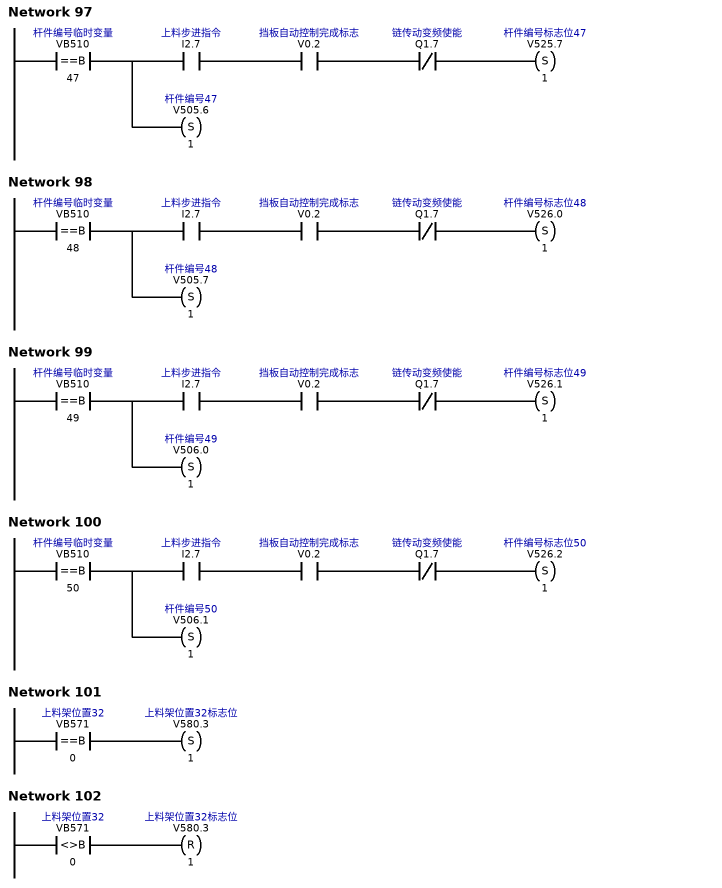
[picture p48: SBR17 networks 97-102]
Network 97
LDB=   杆件编号临时变量:VB510, 47
LPS
A      上料步进指令:I2.7
A      挡板自动控制完成标志:V0.2
AN     链传动变频使能:Q1.7
S      杆件编号标志位47:V525.7, 1
LPP
S      杆件编号47:V505.6, 1
Network 98
LDB=   杆件编号临时变量:VB510, 48
LPS
A      上料步进指令:I2.7
A      挡板自动控制完成标志:V0.2
AN     链传动变频使能:Q1.7
S      杆件编号标志位48:V526.0, 1
LPP
S      杆件编号48:V505.7, 1
Network 99
LDB=   杆件编号临时变量:VB510, 49
LPS
A      上料步进指令:I2.7
A      挡板自动控制完成标志:V0.2
AN     链传动变频使能:Q1.7
S      杆件编号标志位49:V526.1, 1
LPP
S      杆件编号49:V506.0, 1
Network 100
LDB=   杆件编号临时变量:VB510, 50
LPS
A      上料步进指令:I2.7
A      挡板自动控制完成标志:V0.2
AN     链传动变频使能:Q1.7
S      杆件编号标志位50:V526.2, 1
LPP
S      杆件编号50:V506.1, 1
Network 101
LDB=   上料架位置32:VB571, 0
S      上料架位置32标志位:V580.3, 1
Network 102
LDB<>  上料架位置32:VB571, 0
R      上料架位置32标志位:V580.3, 1
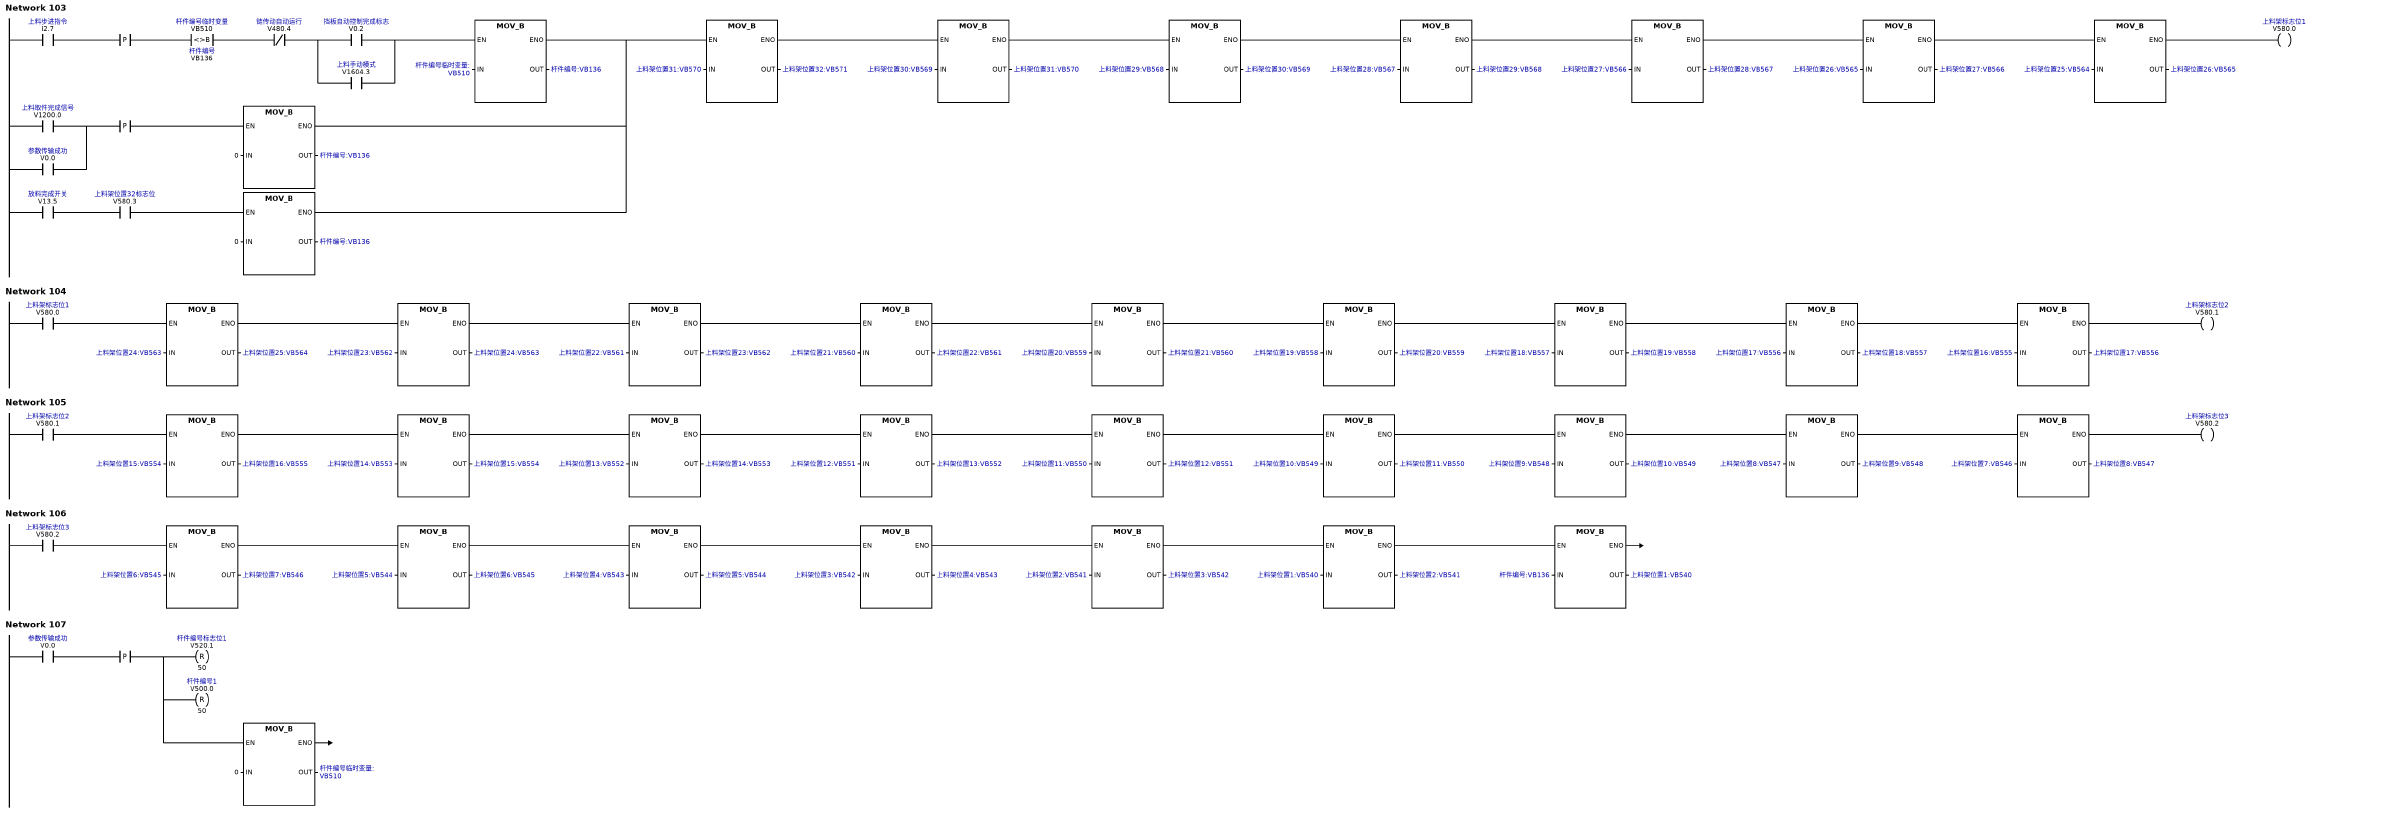
Network 103
LD     上料步进指令:I2.7
EU
AB<>   杆件编号临时变量:VB510, 杆件编号:VB136
AN     链传动自动运行:V480.4
LD     挡板自动控制完成标志:V0.2
O      上料手动模式:V1604.3
ALD
MOVB   杆件编号临时变量:VB510, 杆件编号:VB136
AENO
LD     上料取件完成信号:V1200.0
O      参数传输成功:V0.0
EU
MOVB   0, 杆件编号:VB136
AENO
OLD
LD     放料完成开关:V13.5
A      上料架位置32标志位:V580.3
MOVB   0, 杆件编号:VB136
AENO
OLD
MOVB   上料架位置31:VB570, 上料架位置32:VB571
AENO
MOVB   上料架位置30:VB569, 上料架位置31:VB570
AENO
MOVB   上料架位置29:VB568, 上料架位置30:VB569
AENO
MOVB   上料架位置28:VB567, 上料架位置29:VB568
AENO
MOVB   上料架位置27:VB566, 上料架位置28:VB567
AENO
MOVB   上料架位置26:VB565, 上料架位置27:VB566
AENO
MOVB   上料架位置25:VB564, 上料架位置26:VB565
AENO
=      上料架标志位1:V580.0
Network 104
LD     上料架标志位1:V580.0
MOVB   上料架位置24:VB563, 上料架位置25:VB564
AENO
MOVB   上料架位置23:VB562, 上料架位置24:VB563
AENO
MOVB   上料架位置22:VB561, 上料架位置23:VB562
AENO
MOVB   上料架位置21:VB560, 上料架位置22:VB561
AENO
MOVB   上料架位置20:VB559, 上料架位置21:VB560
AENO
MOVB   上料架位置19:VB558, 上料架位置20:VB559
AENO
MOVB   上料架位置18:VB557, 上料架位置19:VB558
AENO
MOVB   上料架位置17:VB556, 上料架位置18:VB557
AENO
MOVB   上料架位置16:VB555, 上料架位置17:VB556
AENO
=      上料架标志位2:V580.1
Network 105
LD     上料架标志位2:V580.1
MOVB   上料架位置15:VB554, 上料架位置16:VB555
AENO
MOVB   上料架位置14:VB553, 上料架位置15:VB554
AENO
MOVB   上料架位置13:VB552, 上料架位置14:VB553
AENO
MOVB   上料架位置12:VB551, 上料架位置13:VB552
AENO
MOVB   上料架位置11:VB550, 上料架位置12:VB551
AENO
MOVB   上料架位置10:VB549, 上料架位置11:VB550
AENO
MOVB   上料架位置9:VB548, 上料架位置10:VB549
AENO
MOVB   上料架位置8:VB547, 上料架位置9:VB548
AENO
MOVB   上料架位置7:VB546, 上料架位置8:VB547
AENO
=      上料架标志位3:V580.2
Network 106
LD     上料架标志位3:V580.2
MOVB   上料架位置6:VB545, 上料架位置7:VB546
AENO
MOVB   上料架位置5:VB544, 上料架位置6:VB545
AENO
MOVB   上料架位置4:VB543, 上料架位置5:VB544
AENO
MOVB   上料架位置3:VB542, 上料架位置4:VB543
AENO
MOVB   上料架位置2:VB541, 上料架位置3:VB542
AENO
MOVB   上料架位置1:VB540, 上料架位置2:VB541
AENO
MOVB   杆件编号:VB136, 上料架位置1:VB540
Network 107
LD     参数传输成功:V0.0
EU
R      杆件编号标志位1:V520.1, 50
R      杆件编号1:V500.0, 50
MOVB   0, 杆件编号临时变量:VB510
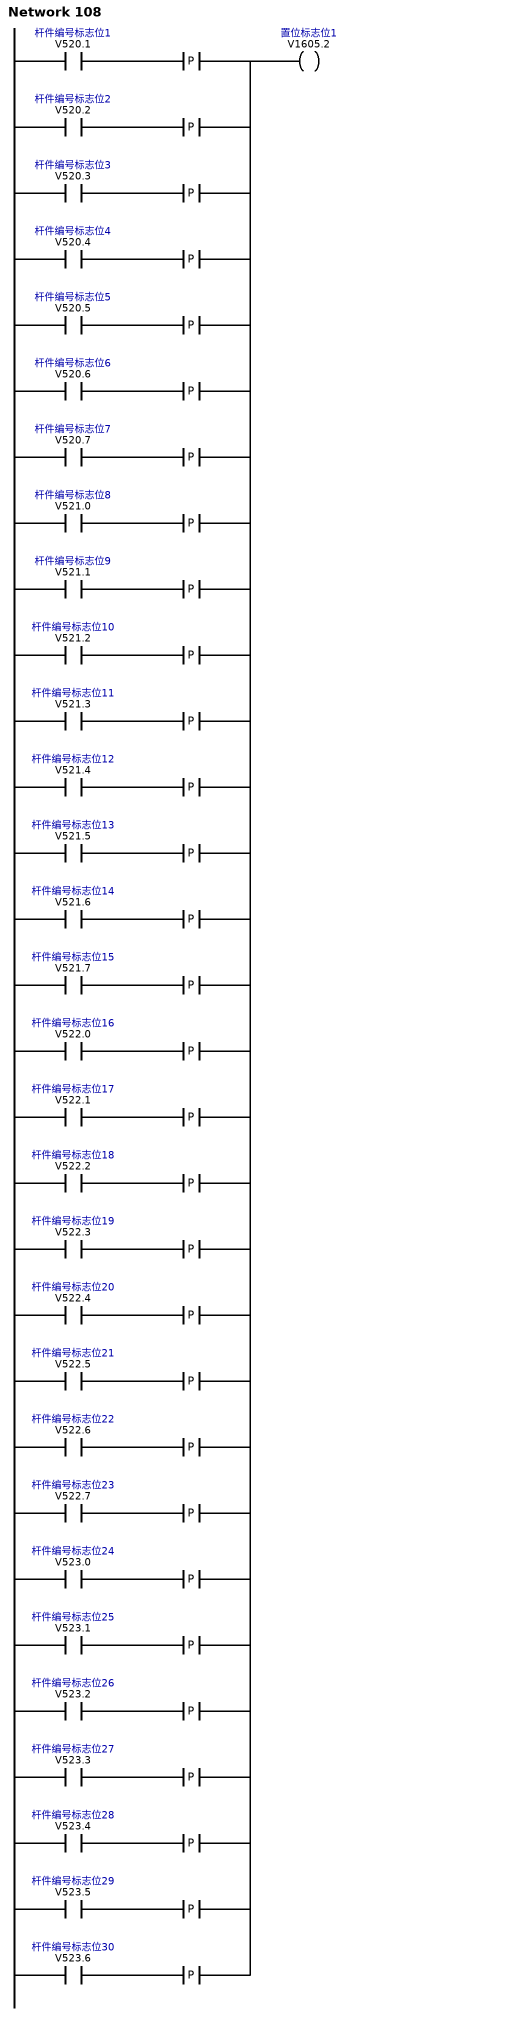
Network 108
LD     杆件编号标志位1:V520.1
EU
LD     杆件编号标志位2:V520.2
EU
OLD
LD     杆件编号标志位3:V520.3
EU
OLD
LD     杆件编号标志位4:V520.4
EU
OLD
LD     杆件编号标志位5:V520.5
EU
OLD
LD     杆件编号标志位6:V520.6
EU
OLD
LD     杆件编号标志位7:V520.7
EU
OLD
LD     杆件编号标志位8:V521.0
EU
OLD
LD     杆件编号标志位9:V521.1
EU
OLD
LD     杆件编号标志位10:V521.2
EU
OLD
LD     杆件编号标志位11:V521.3
EU
OLD
LD     杆件编号标志位12:V521.4
EU
OLD
LD     杆件编号标志位13:V521.5
EU
OLD
LD     杆件编号标志位14:V521.6
EU
OLD
LD     杆件编号标志位15:V521.7
EU
OLD
LD     杆件编号标志位16:V522.0
EU
OLD
LD     杆件编号标志位17:V522.1
EU
OLD
LD     杆件编号标志位18:V522.2
EU
OLD
LD     杆件编号标志位19:V522.3
EU
OLD
LD     杆件编号标志位20:V522.4
EU
OLD
LD     杆件编号标志位21:V522.5
EU
OLD
LD     杆件编号标志位22:V522.6
EU
OLD
LD     杆件编号标志位23:V522.7
EU
OLD
LD     杆件编号标志位24:V523.0
EU
OLD
LD     杆件编号标志位25:V523.1
EU
OLD
LD     杆件编号标志位26:V523.2
EU
OLD
LD     杆件编号标志位27:V523.3
EU
OLD
LD     杆件编号标志位28:V523.4
EU
OLD
LD     杆件编号标志位29:V523.5
EU
OLD
LD     杆件编号标志位30:V523.6
EU
OLD
=      置位标志位1:V1605.2
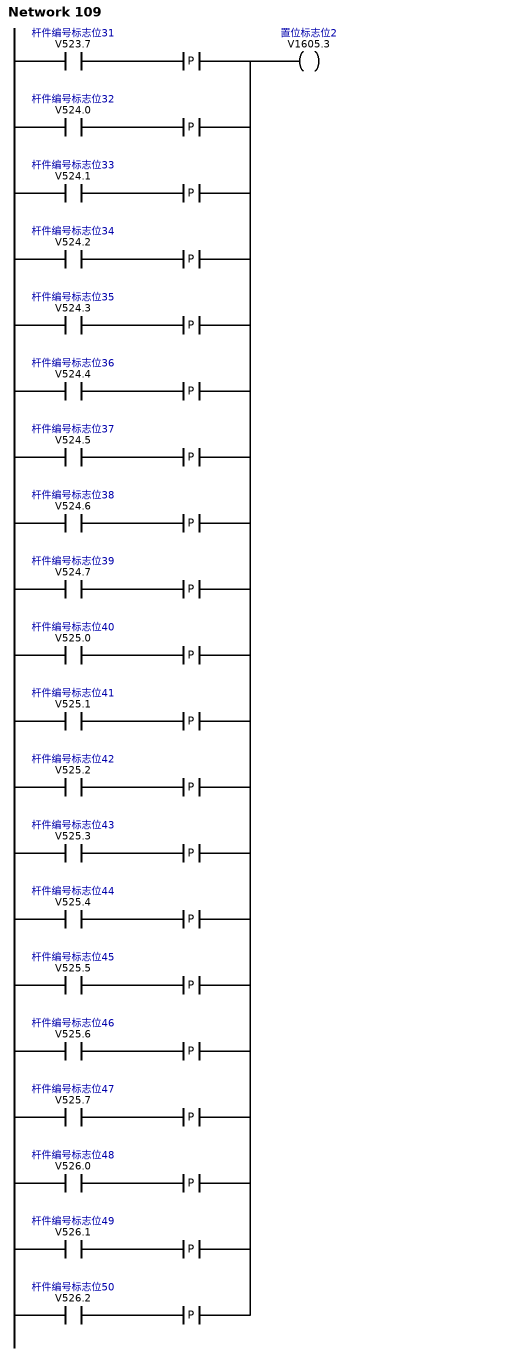
Network 109
LD     杆件编号标志位31:V523.7
EU
LD     杆件编号标志位32:V524.0
EU
OLD
LD     杆件编号标志位33:V524.1
EU
OLD
LD     杆件编号标志位34:V524.2
EU
OLD
LD     杆件编号标志位35:V524.3
EU
OLD
LD     杆件编号标志位36:V524.4
EU
OLD
LD     杆件编号标志位37:V524.5
EU
OLD
LD     杆件编号标志位38:V524.6
EU
OLD
LD     杆件编号标志位39:V524.7
EU
OLD
LD     杆件编号标志位40:V525.0
EU
OLD
LD     杆件编号标志位41:V525.1
EU
OLD
LD     杆件编号标志位42:V525.2
EU
OLD
LD     杆件编号标志位43:V525.3
EU
OLD
LD     杆件编号标志位44:V525.4
EU
OLD
LD     杆件编号标志位45:V525.5
EU
OLD
LD     杆件编号标志位46:V525.6
EU
OLD
LD     杆件编号标志位47:V525.7
EU
OLD
LD     杆件编号标志位48:V526.0
EU
OLD
LD     杆件编号标志位49:V526.1
EU
OLD
LD     杆件编号标志位50:V526.2
EU
OLD
=      置位标志位2:V1605.3
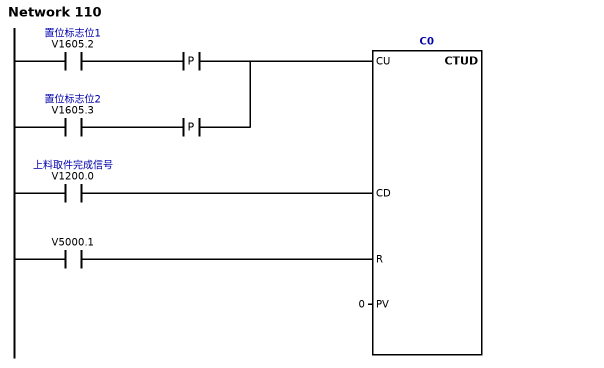
Network 110
LD     置位标志位1:V1605.2
EU
LD     置位标志位2:V1605.3
EU
OLD
LD     上料取件完成信号:V1200.0
LD     V5000.1
CTUD   C0, 0
END_SUBROUTINE_BLOCK

SUBROUTINE_BLOCK 冷却电机手动控制:SBR18
TITLE=子程序注释
BEGIN
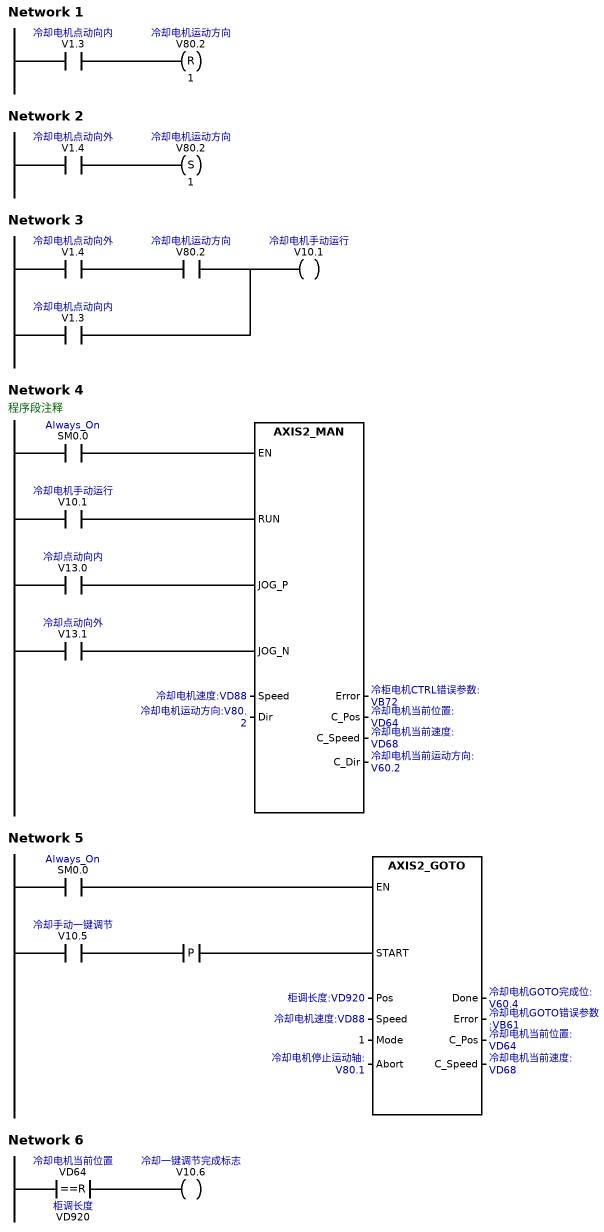
Network 1
LD     冷却电机点动向内:V1.3
R      冷却电机运动方向:V80.2, 1
Network 2
LD     冷却电机点动向外:V1.4
S      冷却电机运动方向:V80.2, 1
Network 3
LD     冷却电机点动向外:V1.4
A      冷却电机运动方向:V80.2
O      冷却电机点动向内:V1.3
=      冷却电机手动运行:V10.1
Network 4
// 程序段注释
LD     Always_On:SM0.0
=      L60.0
LD     冷却电机手动运行:V10.1
=      L63.7
LD     冷却点动向内:V13.0
=      L63.6
LD     冷却点动向外:V13.1
=      L63.5
LD     L60.0
CALL   AXIS2_MAN:SBR11, L63.7, L63.6, L63.5, 冷却电机速度:VD88, 冷却电机运动方向:V80.2, 冷柜电机CTRL错误参数:VB72, 冷却电机当前位置:VD64, 冷却电机当前速度:VD68, 冷却电机当前运动方向:V60.2
Network 5
LD     Always_On:SM0.0
=      L60.0
LD     冷却手动一键调节:V10.5
EU
=      L63.7
LD     L60.0
CALL   AXIS2_GOTO:SBR12, L63.7, 柜调长度:VD920, 冷却电机速度:VD88, 1, 冷却电机停止运动轴:V80.1, 冷却电机GOTO完成位:V60.4, 冷却电机GOTO错误参数:VB61, 冷却电机当前位置:VD64, 冷却电机当前速度:VD68
Network 6
LDR=   冷却电机当前位置:VD64, 柜调长度:VD920
=      冷却一键调节完成标志:V10.6
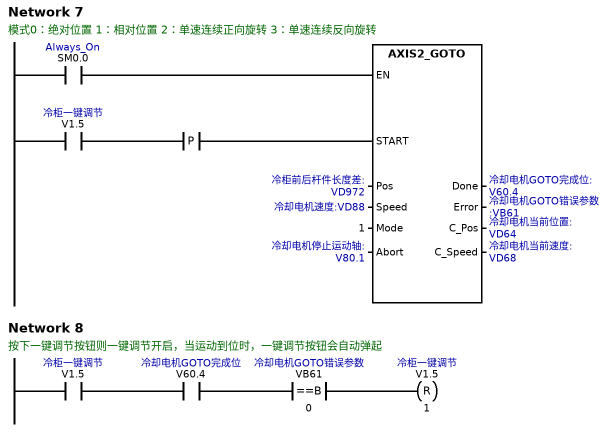
Network 7
// 模式0：绝对位置 1：相对位置 2：单速连续正向旋转 3：单速连续反向旋转
LD     Always_On:SM0.0
=      L60.0
LD     冷柜一键调节:V1.5
EU
=      L63.7
LD     L60.0
CALL   AXIS2_GOTO:SBR12, L63.7, 冷柜前后杆件长度差:VD972, 冷却电机速度:VD88, 1, 冷却电机停止运动轴:V80.1, 冷却电机GOTO完成位:V60.4, 冷却电机GOTO错误参数:VB61, 冷却电机当前位置:VD64, 冷却电机当前速度:VD68
Network 8
// 按下一键调节按钮则一键调节开启，当运动到位时，一键调节按钮会自动弹起
LD     冷柜一键调节:V1.5
A      冷却电机GOTO完成位:V60.4
AB=    冷却电机GOTO错误参数:VB61, 0
R      冷柜一键调节:V1.5, 1
END_SUBROUTINE_BLOCK

SUBROUTINE_BLOCK 链传动电机控制:SBR19
TITLE=子程序注释
BEGIN
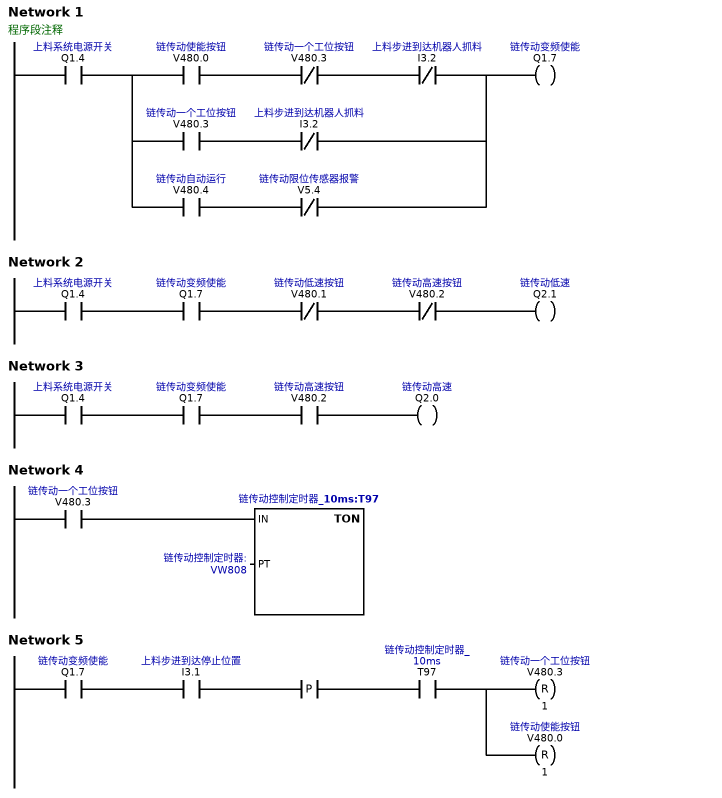
Network 1
// 程序段注释
LD     上料系统电源开关:Q1.4
LD     链传动使能按钮:V480.0
AN     链传动一个工位按钮:V480.3
AN     上料步进到达机器人抓料:I3.2
LD     链传动一个工位按钮:V480.3
AN     上料步进到达机器人抓料:I3.2
OLD
LD     链传动自动运行:V480.4
AN     链传动限位传感器报警:V5.4
OLD
ALD
=      链传动变频使能:Q1.7
Network 2
LD     上料系统电源开关:Q1.4
A      链传动变频使能:Q1.7
AN     链传动低速按钮:V480.1
AN     链传动高速按钮:V480.2
=      链传动低速:Q2.1
Network 3
LD     上料系统电源开关:Q1.4
A      链传动变频使能:Q1.7
A      链传动高速按钮:V480.2
=      链传动高速:Q2.0
Network 4
LD     链传动一个工位按钮:V480.3
TON    链传动控制定时器_10ms:T97, 链传动控制定时器:VW808
Network 5
LD     链传动变频使能:Q1.7
A      上料步进到达停止位置:I3.1
EU
A      链传动控制定时器_10ms:T97
R      链传动一个工位按钮:V480.3, 1
R      链传动使能按钮:V480.0, 1
END_SUBROUTINE_BLOCK

SUBROUTINE_BLOCK 数据初始化:SBR20
TITLE=子程序注释
BEGIN
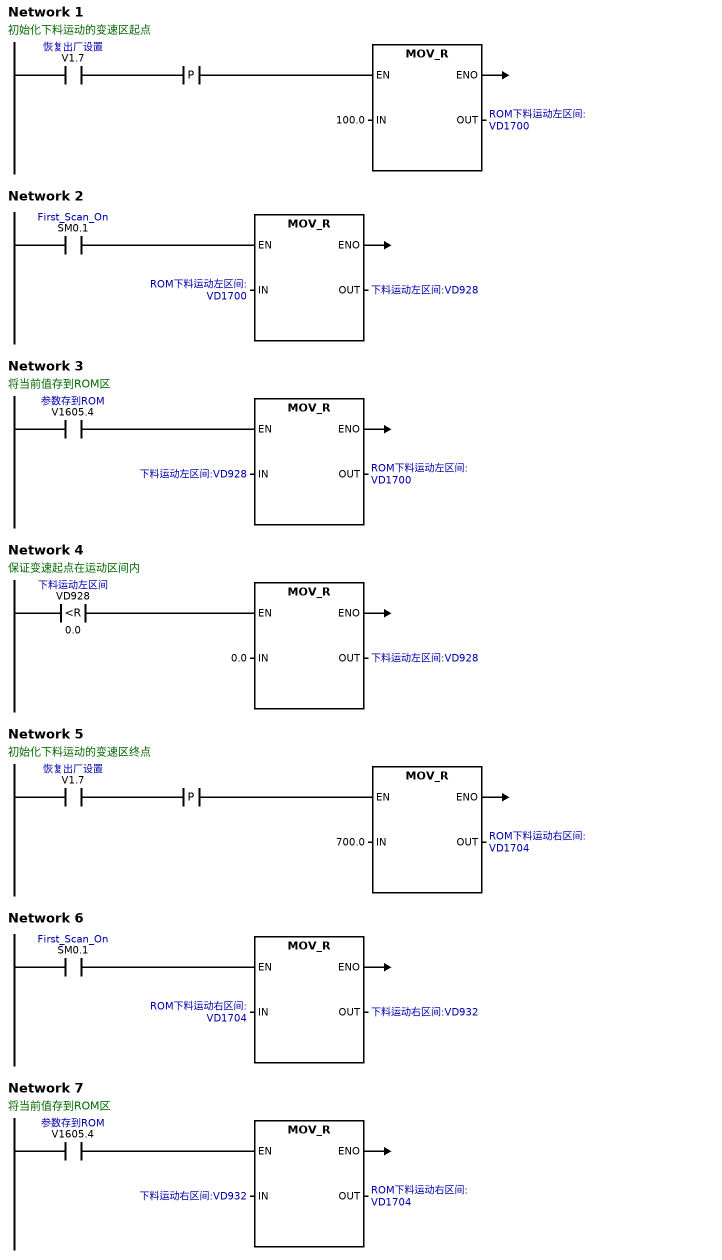
Network 1
// 初始化下料运动的变速区起点
LD     恢复出厂设置:V1.7
EU
MOVR   100.0, ROM下料运动左区间:VD1700
Network 2
LD     First_Scan_On:SM0.1
MOVR   ROM下料运动左区间:VD1700, 下料运动左区间:VD928
Network 3
// 将当前值存到ROM区
LD     参数存到ROM:V1605.4
MOVR   下料运动左区间:VD928, ROM下料运动左区间:VD1700
Network 4
// 保证变速起点在运动区间内
LDR<   下料运动左区间:VD928, 0.0
MOVR   0.0, 下料运动左区间:VD928
Network 5
// 初始化下料运动的变速区终点
LD     恢复出厂设置:V1.7
EU
MOVR   700.0, ROM下料运动右区间:VD1704
Network 6
LD     First_Scan_On:SM0.1
MOVR   ROM下料运动右区间:VD1704, 下料运动右区间:VD932
Network 7
// 将当前值存到ROM区
LD     参数存到ROM:V1605.4
MOVR   下料运动右区间:VD932, ROM下料运动右区间:VD1704
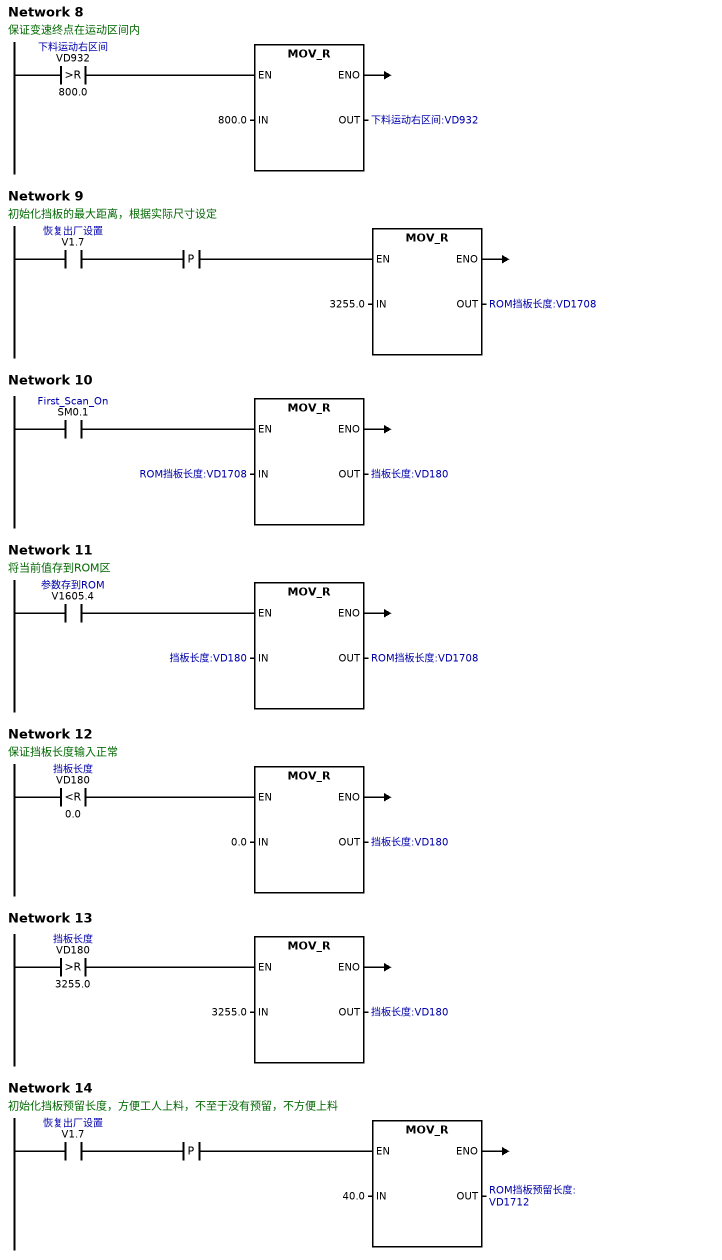
Network 8
// 保证变速终点在运动区间内
LDR>   下料运动右区间:VD932, 800.0
MOVR   800.0, 下料运动右区间:VD932
Network 9
// 初始化挡板的最大距离，根据实际尺寸设定
LD     恢复出厂设置:V1.7
EU
MOVR   3255.0, ROM挡板长度:VD1708
Network 10
LD     First_Scan_On:SM0.1
MOVR   ROM挡板长度:VD1708, 挡板长度:VD180
Network 11
// 将当前值存到ROM区
LD     参数存到ROM:V1605.4
MOVR   挡板长度:VD180, ROM挡板长度:VD1708
Network 12
// 保证挡板长度输入正常
LDR<   挡板长度:VD180, 0.0
MOVR   0.0, 挡板长度:VD180
Network 13
LDR>   挡板长度:VD180, 3255.0
MOVR   3255.0, 挡板长度:VD180
Network 14
// 初始化挡板预留长度，方便工人上料，不至于没有预留，不方便上料
LD     恢复出厂设置:V1.7
EU
MOVR   40.0, ROM挡板预留长度:VD1712
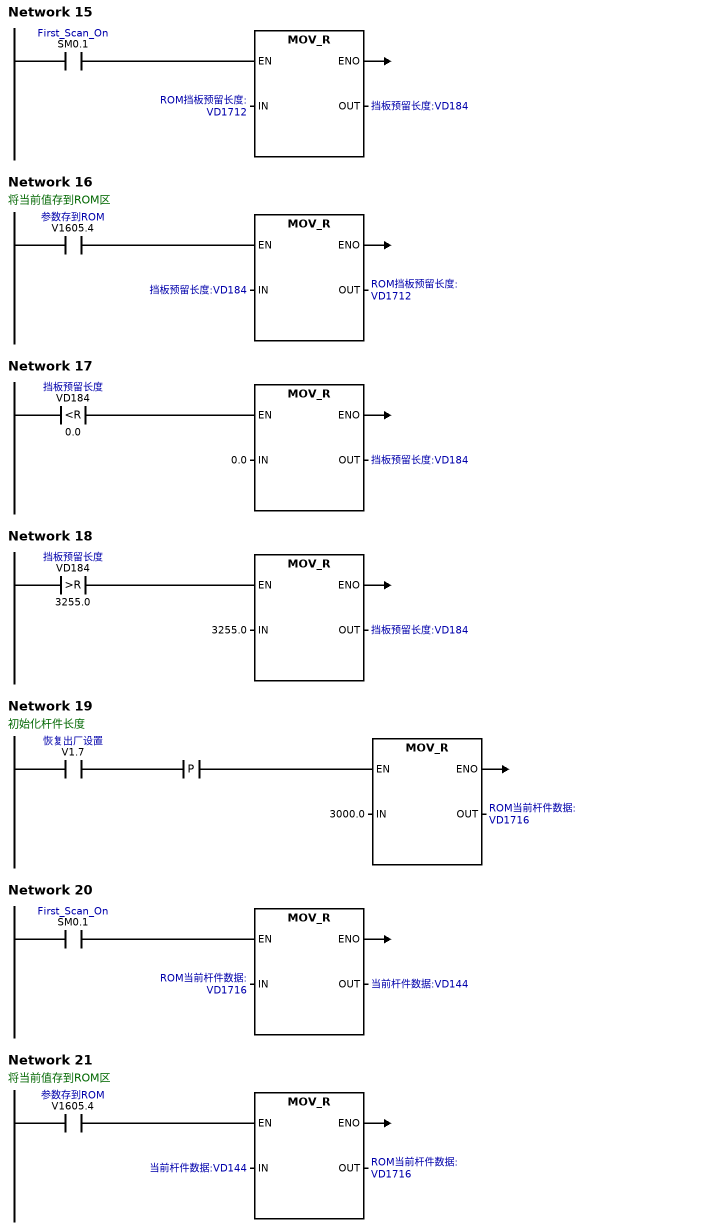
Network 15
LD     First_Scan_On:SM0.1
MOVR   ROM挡板预留长度:VD1712, 挡板预留长度:VD184
Network 16
// 将当前值存到ROM区
LD     参数存到ROM:V1605.4
MOVR   挡板预留长度:VD184, ROM挡板预留长度:VD1712
Network 17
LDR<   挡板预留长度:VD184, 0.0
MOVR   0.0, 挡板预留长度:VD184
Network 18
LDR>   挡板预留长度:VD184, 3255.0
MOVR   3255.0, 挡板预留长度:VD184
Network 19
// 初始化杆件长度
LD     恢复出厂设置:V1.7
EU
MOVR   3000.0, ROM当前杆件数据:VD1716
Network 20
LD     First_Scan_On:SM0.1
MOVR   ROM当前杆件数据:VD1716, 当前杆件数据:VD144
Network 21
// 将当前值存到ROM区
LD     参数存到ROM:V1605.4
MOVR   当前杆件数据:VD144, ROM当前杆件数据:VD1716
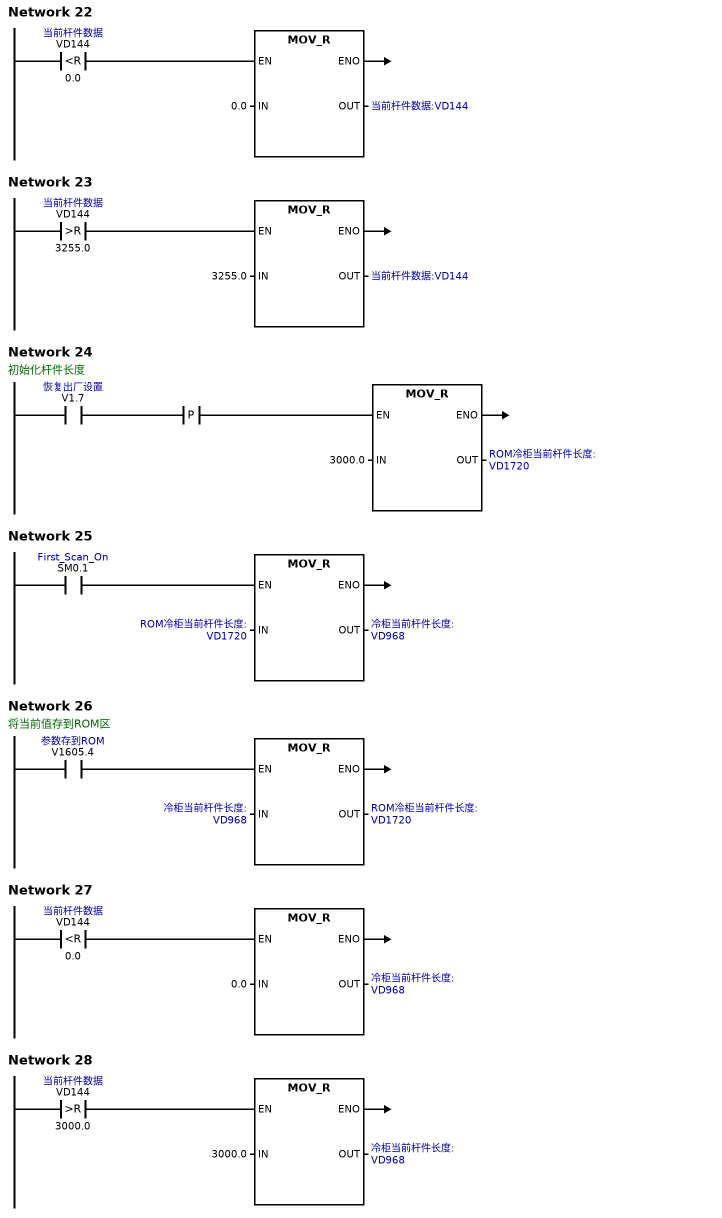
Network 22
LDR<   当前杆件数据:VD144, 0.0
MOVR   0.0, 当前杆件数据:VD144
Network 23
LDR>   当前杆件数据:VD144, 3255.0
MOVR   3255.0, 当前杆件数据:VD144
Network 24
// 初始化杆件长度
LD     恢复出厂设置:V1.7
EU
MOVR   3000.0, ROM冷柜当前杆件长度:VD1720
Network 25
LD     First_Scan_On:SM0.1
MOVR   ROM冷柜当前杆件长度:VD1720, 冷柜当前杆件长度:VD968
Network 26
// 将当前值存到ROM区
LD     参数存到ROM:V1605.4
MOVR   冷柜当前杆件长度:VD968, ROM冷柜当前杆件长度:VD1720
Network 27
LDR<   当前杆件数据:VD144, 0.0
MOVR   0.0, 冷柜当前杆件长度:VD968
Network 28
LDR>   当前杆件数据:VD144, 3000.0
MOVR   3000.0, 冷柜当前杆件长度:VD968
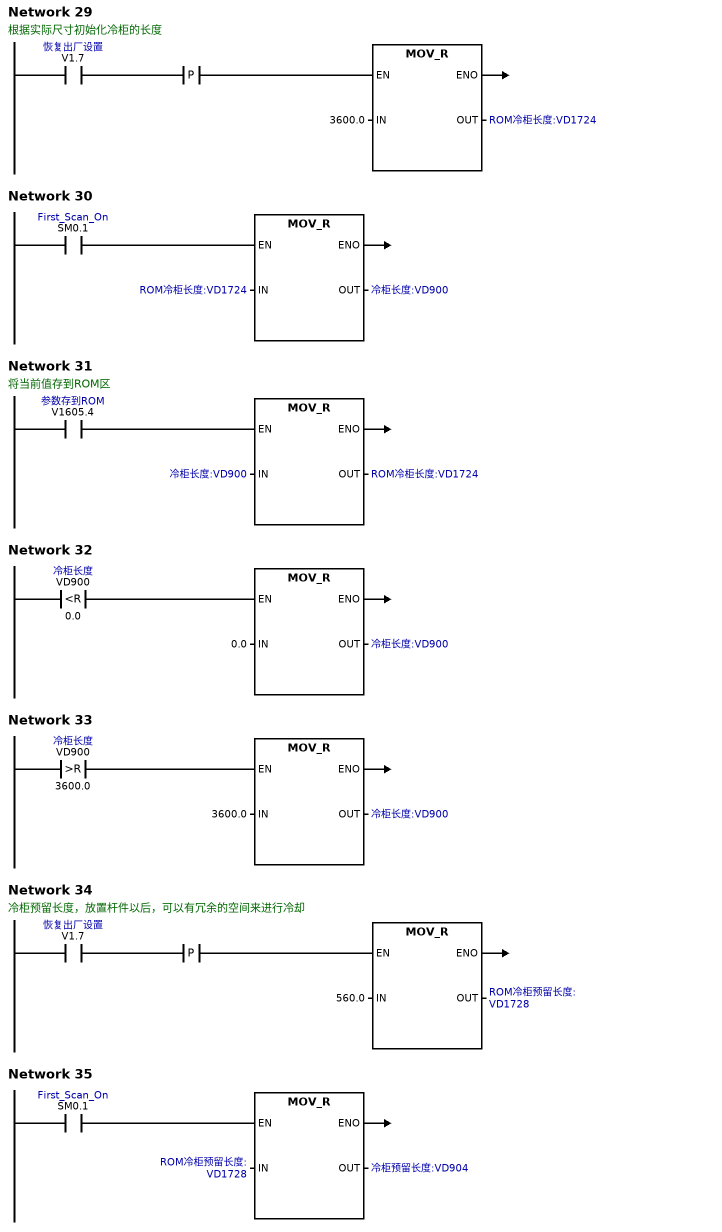
Network 29
// 根据实际尺寸初始化冷柜的长度
LD     恢复出厂设置:V1.7
EU
MOVR   3600.0, ROM冷柜长度:VD1724
Network 30
LD     First_Scan_On:SM0.1
MOVR   ROM冷柜长度:VD1724, 冷柜长度:VD900
Network 31
// 将当前值存到ROM区
LD     参数存到ROM:V1605.4
MOVR   冷柜长度:VD900, ROM冷柜长度:VD1724
Network 32
LDR<   冷柜长度:VD900, 0.0
MOVR   0.0, 冷柜长度:VD900
Network 33
LDR>   冷柜长度:VD900, 3600.0
MOVR   3600.0, 冷柜长度:VD900
Network 34
// 冷柜预留长度，放置杆件以后，可以有冗余的空间来进行冷却
LD     恢复出厂设置:V1.7
EU
MOVR   560.0, ROM冷柜预留长度:VD1728
Network 35
LD     First_Scan_On:SM0.1
MOVR   ROM冷柜预留长度:VD1728, 冷柜预留长度:VD904
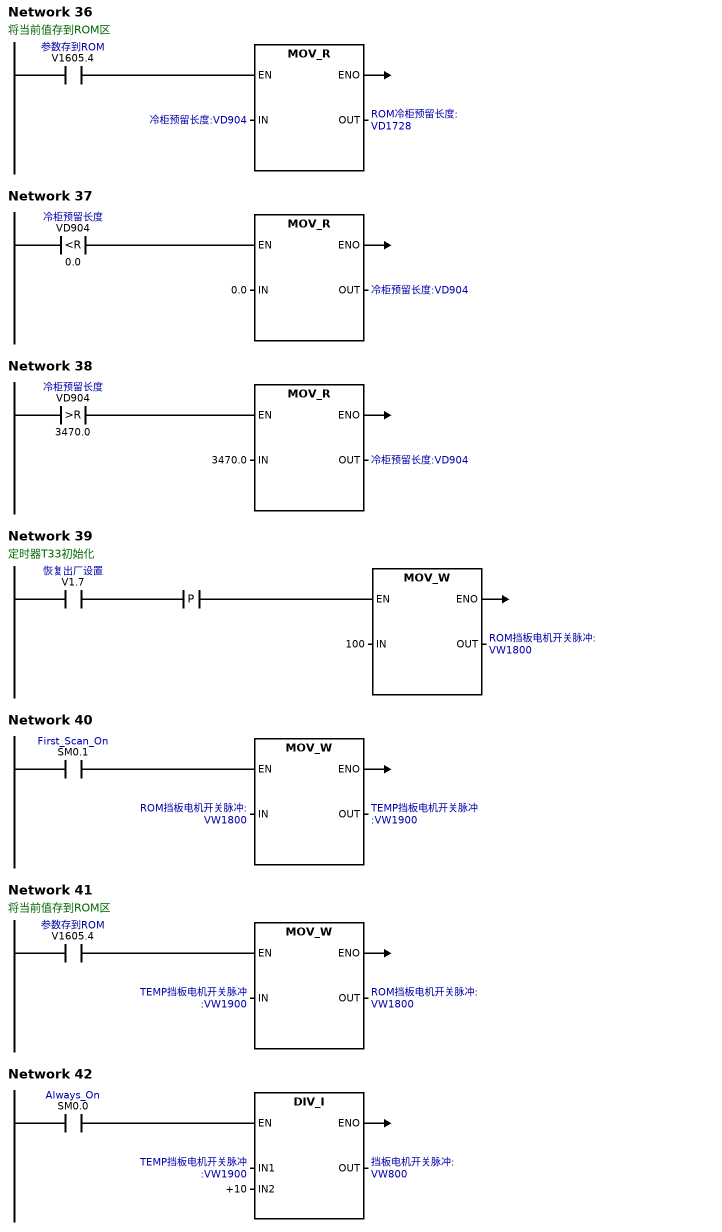
Network 36
// 将当前值存到ROM区
LD     参数存到ROM:V1605.4
MOVR   冷柜预留长度:VD904, ROM冷柜预留长度:VD1728
Network 37
LDR<   冷柜预留长度:VD904, 0.0
MOVR   0.0, 冷柜预留长度:VD904
Network 38
LDR>   冷柜预留长度:VD904, 3470.0
MOVR   3470.0, 冷柜预留长度:VD904
Network 39
// 定时器T33初始化
LD     恢复出厂设置:V1.7
EU
MOVW   100, ROM挡板电机开关脉冲:VW1800
Network 40
LD     First_Scan_On:SM0.1
MOVW   ROM挡板电机开关脉冲:VW1800, TEMP挡板电机开关脉冲:VW1900
Network 41
// 将当前值存到ROM区
LD     参数存到ROM:V1605.4
MOVW   TEMP挡板电机开关脉冲:VW1900, ROM挡板电机开关脉冲:VW1800
Network 42
LD     Always_On:SM0.0
MOVW   TEMP挡板电机开关脉冲:VW1900, 挡板电机开关脉冲:VW800
/I     +10, 挡板电机开关脉冲:VW800
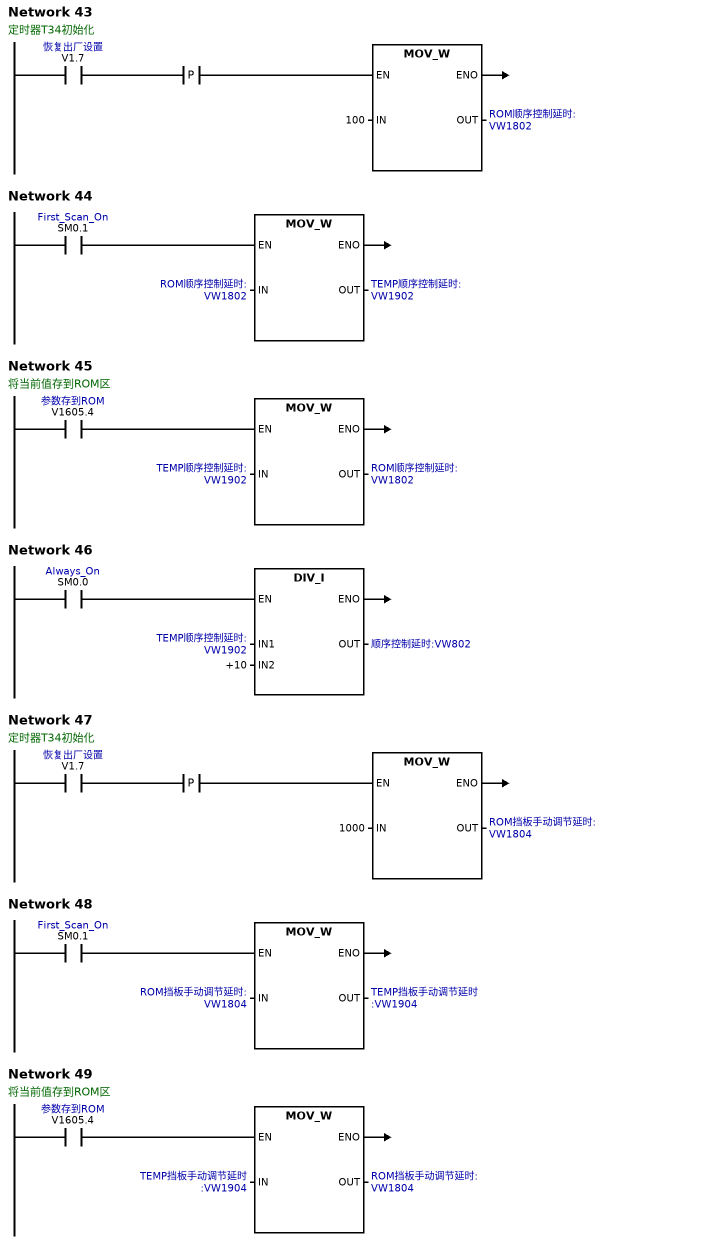
Network 43
// 定时器T34初始化
LD     恢复出厂设置:V1.7
EU
MOVW   100, ROM顺序控制延时:VW1802
Network 44
LD     First_Scan_On:SM0.1
MOVW   ROM顺序控制延时:VW1802, TEMP顺序控制延时:VW1902
Network 45
// 将当前值存到ROM区
LD     参数存到ROM:V1605.4
MOVW   TEMP顺序控制延时:VW1902, ROM顺序控制延时:VW1802
Network 46
LD     Always_On:SM0.0
MOVW   TEMP顺序控制延时:VW1902, 顺序控制延时:VW802
/I     +10, 顺序控制延时:VW802
Network 47
// 定时器T34初始化
LD     恢复出厂设置:V1.7
EU
MOVW   1000, ROM挡板手动调节延时:VW1804
Network 48
LD     First_Scan_On:SM0.1
MOVW   ROM挡板手动调节延时:VW1804, TEMP挡板手动调节延时:VW1904
Network 49
// 将当前值存到ROM区
LD     参数存到ROM:V1605.4
MOVW   TEMP挡板手动调节延时:VW1904, ROM挡板手动调节延时:VW1804
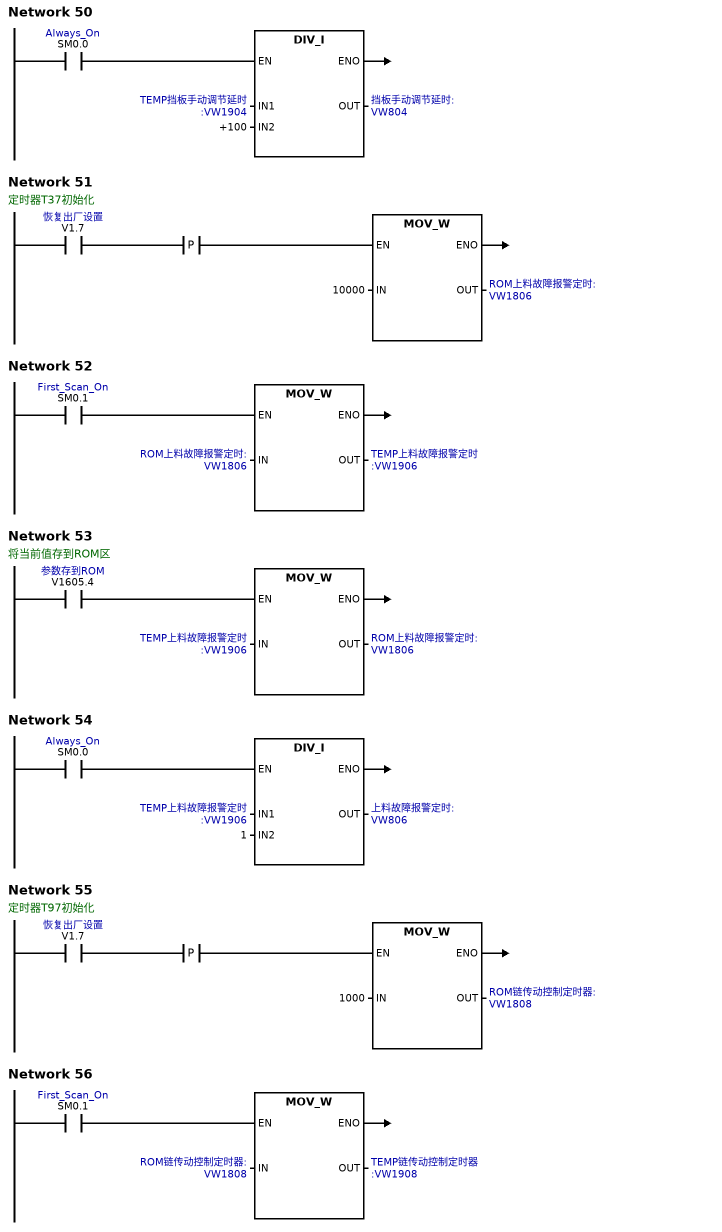
Network 50
LD     Always_On:SM0.0
MOVW   TEMP挡板手动调节延时:VW1904, 挡板手动调节延时:VW804
/I     +100, 挡板手动调节延时:VW804
Network 51
// 定时器T37初始化
LD     恢复出厂设置:V1.7
EU
MOVW   10000, ROM上料故障报警定时:VW1806
Network 52
LD     First_Scan_On:SM0.1
MOVW   ROM上料故障报警定时:VW1806, TEMP上料故障报警定时:VW1906
Network 53
// 将当前值存到ROM区
LD     参数存到ROM:V1605.4
MOVW   TEMP上料故障报警定时:VW1906, ROM上料故障报警定时:VW1806
Network 54
LD     Always_On:SM0.0
MOVW   TEMP上料故障报警定时:VW1906, 上料故障报警定时:VW806
/I     1, 上料故障报警定时:VW806
Network 55
// 定时器T97初始化
LD     恢复出厂设置:V1.7
EU
MOVW   1000, ROM链传动控制定时器:VW1808
Network 56
LD     First_Scan_On:SM0.1
MOVW   ROM链传动控制定时器:VW1808, TEMP链传动控制定时器:VW1908
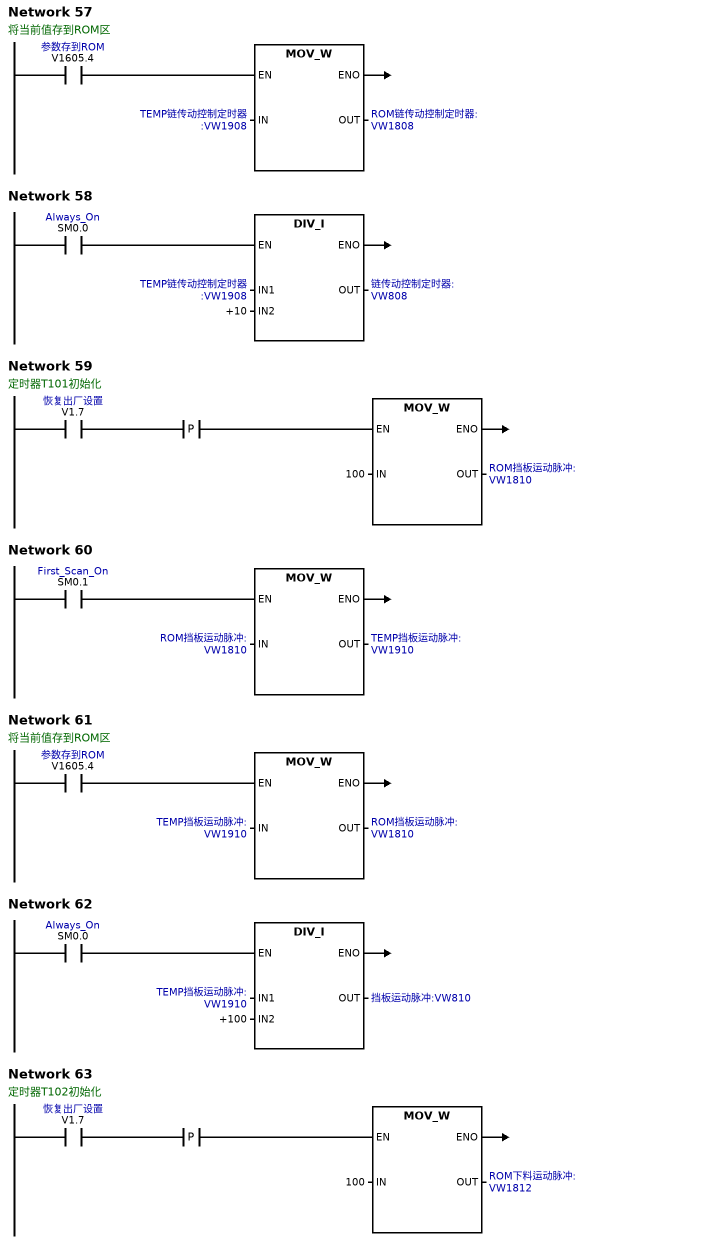
Network 57
// 将当前值存到ROM区
LD     参数存到ROM:V1605.4
MOVW   TEMP链传动控制定时器:VW1908, ROM链传动控制定时器:VW1808
Network 58
LD     Always_On:SM0.0
MOVW   TEMP链传动控制定时器:VW1908, 链传动控制定时器:VW808
/I     +10, 链传动控制定时器:VW808
Network 59
// 定时器T101初始化
LD     恢复出厂设置:V1.7
EU
MOVW   100, ROM挡板运动脉冲:VW1810
Network 60
LD     First_Scan_On:SM0.1
MOVW   ROM挡板运动脉冲:VW1810, TEMP挡板运动脉冲:VW1910
Network 61
// 将当前值存到ROM区
LD     参数存到ROM:V1605.4
MOVW   TEMP挡板运动脉冲:VW1910, ROM挡板运动脉冲:VW1810
Network 62
LD     Always_On:SM0.0
MOVW   TEMP挡板运动脉冲:VW1910, 挡板运动脉冲:VW810
/I     +100, 挡板运动脉冲:VW810
Network 63
// 定时器T102初始化
LD     恢复出厂设置:V1.7
EU
MOVW   100, ROM下料运动脉冲:VW1812
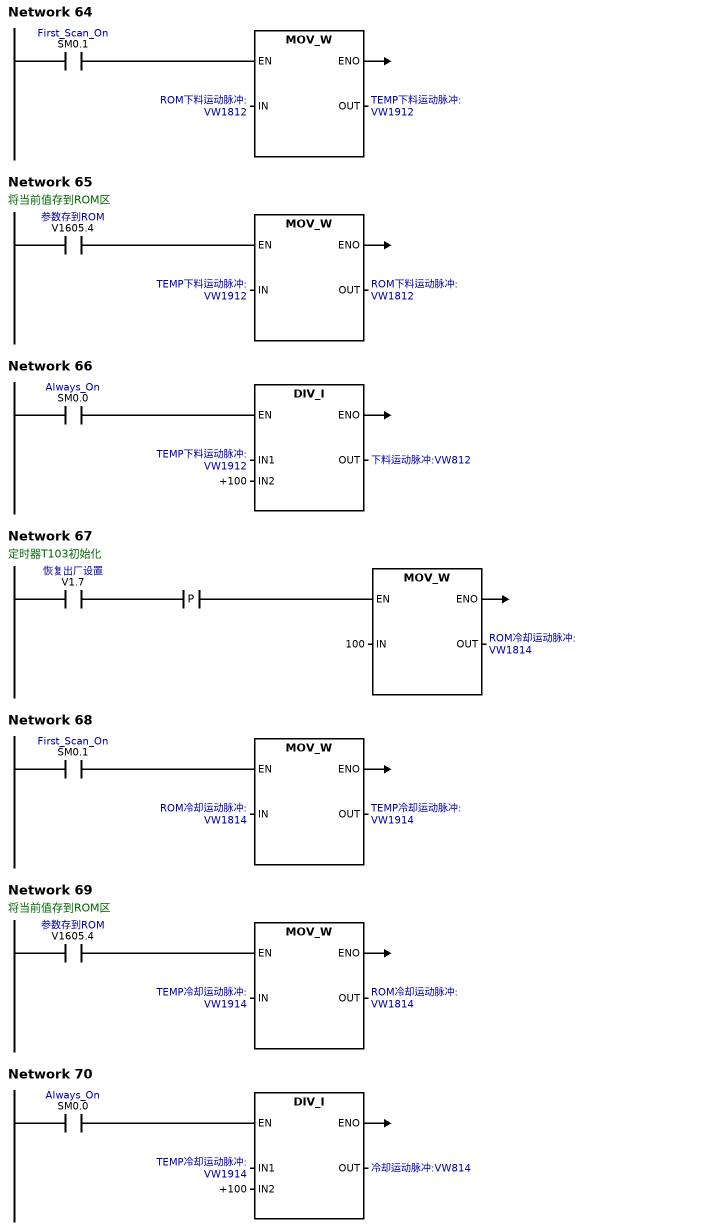
Network 64
LD     First_Scan_On:SM0.1
MOVW   ROM下料运动脉冲:VW1812, TEMP下料运动脉冲:VW1912
Network 65
// 将当前值存到ROM区
LD     参数存到ROM:V1605.4
MOVW   TEMP下料运动脉冲:VW1912, ROM下料运动脉冲:VW1812
Network 66
LD     Always_On:SM0.0
MOVW   TEMP下料运动脉冲:VW1912, 下料运动脉冲:VW812
/I     +100, 下料运动脉冲:VW812
Network 67
// 定时器T103初始化
LD     恢复出厂设置:V1.7
EU
MOVW   100, ROM冷却运动脉冲:VW1814
Network 68
LD     First_Scan_On:SM0.1
MOVW   ROM冷却运动脉冲:VW1814, TEMP冷却运动脉冲:VW1914
Network 69
// 将当前值存到ROM区
LD     参数存到ROM:V1605.4
MOVW   TEMP冷却运动脉冲:VW1914, ROM冷却运动脉冲:VW1814
Network 70
LD     Always_On:SM0.0
MOVW   TEMP冷却运动脉冲:VW1914, 冷却运动脉冲:VW814
/I     +100, 冷却运动脉冲:VW814
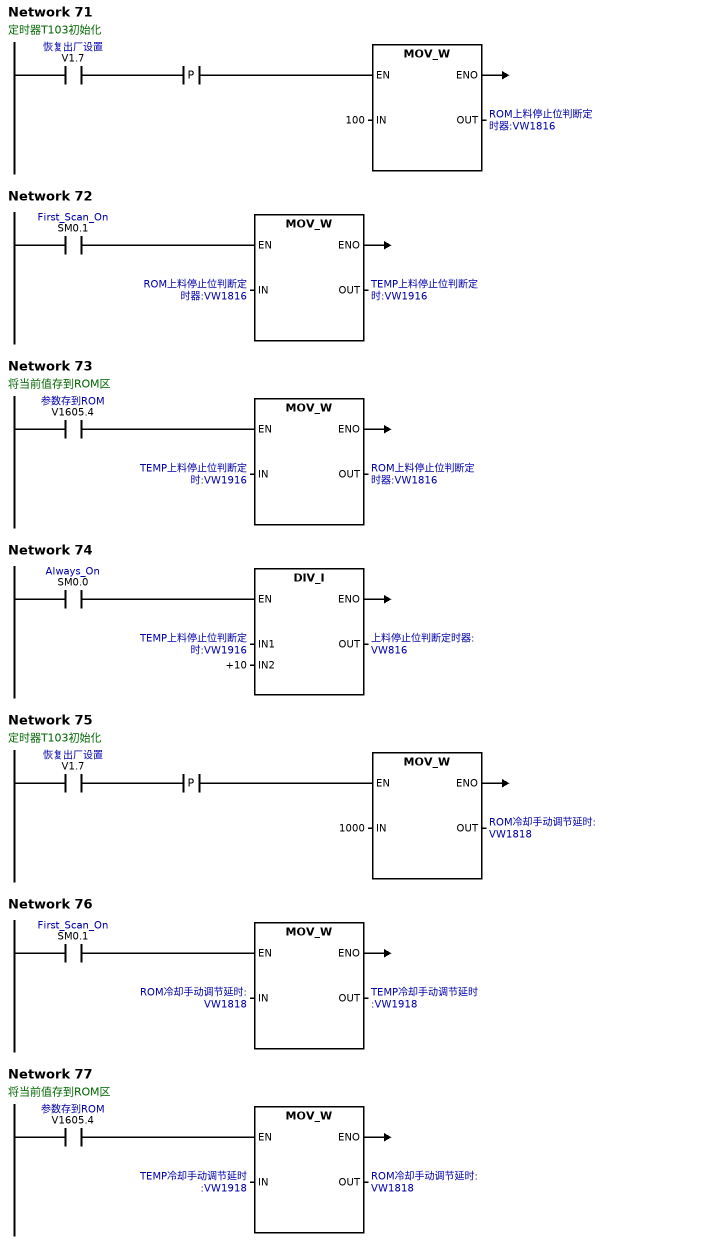
Network 71
// 定时器T103初始化
LD     恢复出厂设置:V1.7
EU
MOVW   100, ROM上料停止位判断定时器:VW1816
Network 72
LD     First_Scan_On:SM0.1
MOVW   ROM上料停止位判断定时器:VW1816, TEMP上料停止位判断定时:VW1916
Network 73
// 将当前值存到ROM区
LD     参数存到ROM:V1605.4
MOVW   TEMP上料停止位判断定时:VW1916, ROM上料停止位判断定时器:VW1816
Network 74
LD     Always_On:SM0.0
MOVW   TEMP上料停止位判断定时:VW1916, 上料停止位判断定时器:VW816
/I     +10, 上料停止位判断定时器:VW816
Network 75
// 定时器T103初始化
LD     恢复出厂设置:V1.7
EU
MOVW   1000, ROM冷却手动调节延时:VW1818
Network 76
LD     First_Scan_On:SM0.1
MOVW   ROM冷却手动调节延时:VW1818, TEMP冷却手动调节延时:VW1918
Network 77
// 将当前值存到ROM区
LD     参数存到ROM:V1605.4
MOVW   TEMP冷却手动调节延时:VW1918, ROM冷却手动调节延时:VW1818
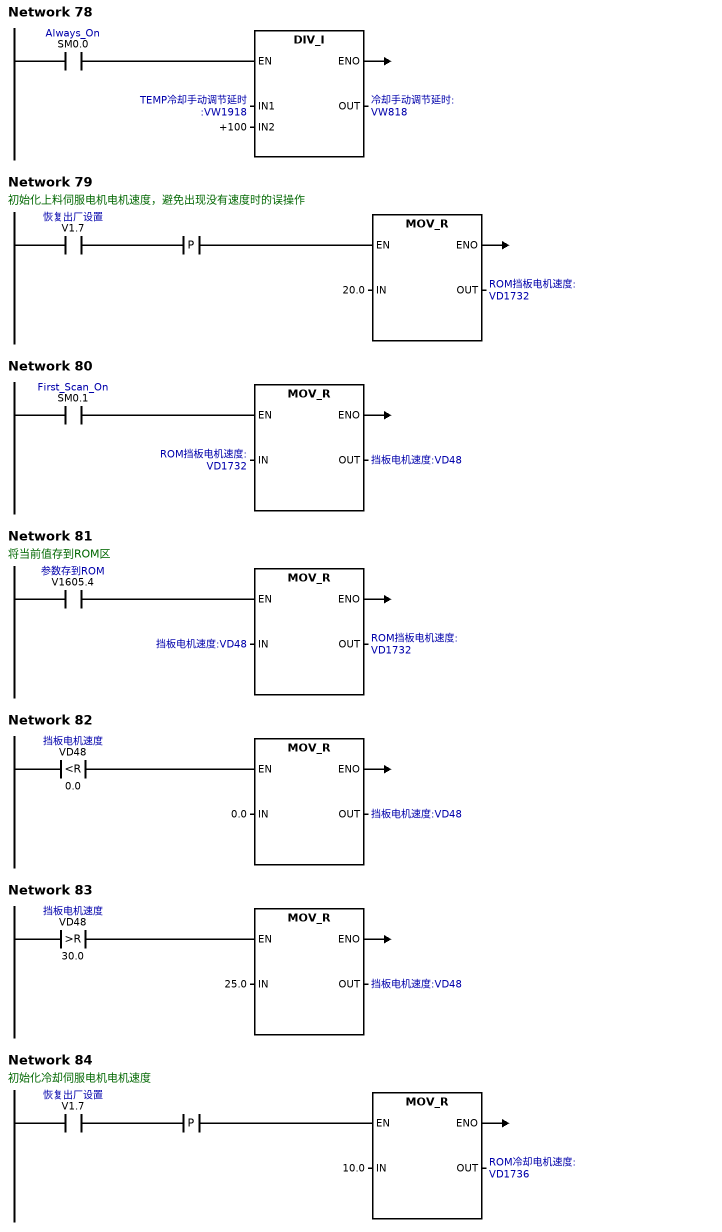
Network 78
LD     Always_On:SM0.0
MOVW   TEMP冷却手动调节延时:VW1918, 冷却手动调节延时:VW818
/I     +100, 冷却手动调节延时:VW818
Network 79
// 初始化上料伺服电机电机速度，避免出现没有速度时的误操作
LD     恢复出厂设置:V1.7
EU
MOVR   20.0, ROM挡板电机速度:VD1732
Network 80
LD     First_Scan_On:SM0.1
MOVR   ROM挡板电机速度:VD1732, 挡板电机速度:VD48
Network 81
// 将当前值存到ROM区
LD     参数存到ROM:V1605.4
MOVR   挡板电机速度:VD48, ROM挡板电机速度:VD1732
Network 82
LDR<   挡板电机速度:VD48, 0.0
MOVR   0.0, 挡板电机速度:VD48
Network 83
LDR>   挡板电机速度:VD48, 30.0
MOVR   25.0, 挡板电机速度:VD48
Network 84
// 初始化冷却伺服电机电机速度
LD     恢复出厂设置:V1.7
EU
MOVR   10.0, ROM冷却电机速度:VD1736
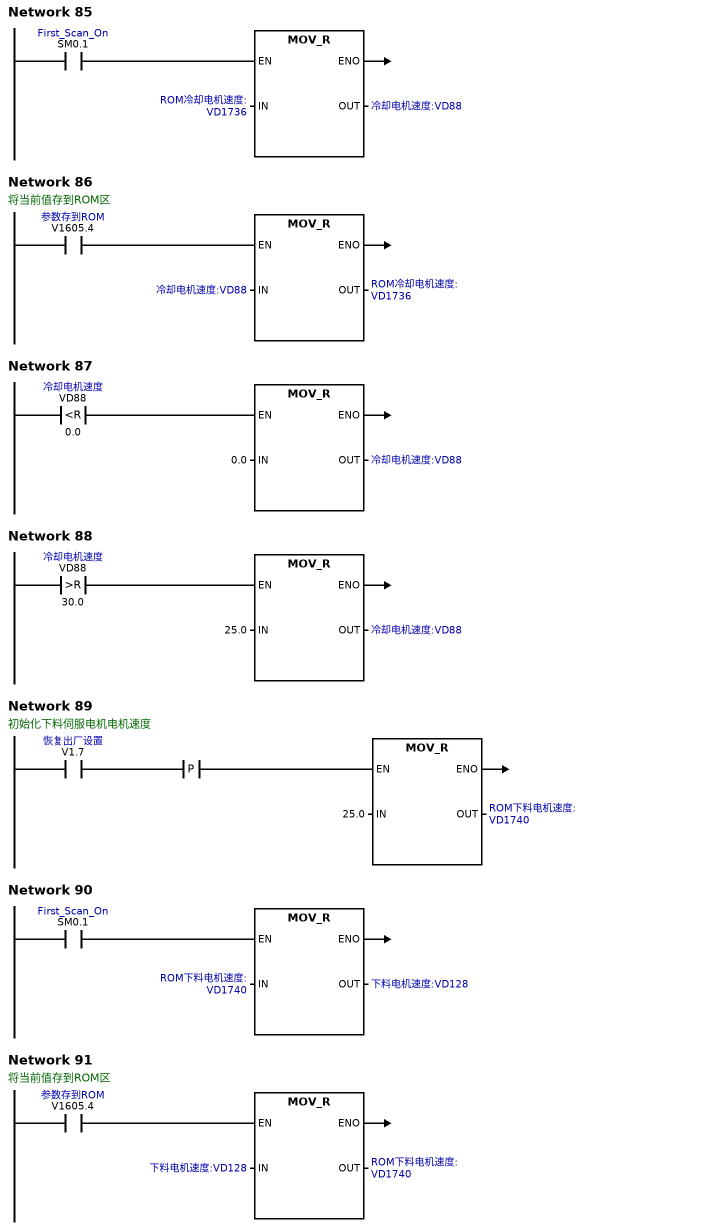
Network 85
LD     First_Scan_On:SM0.1
MOVR   ROM冷却电机速度:VD1736, 冷却电机速度:VD88
Network 86
// 将当前值存到ROM区
LD     参数存到ROM:V1605.4
MOVR   冷却电机速度:VD88, ROM冷却电机速度:VD1736
Network 87
LDR<   冷却电机速度:VD88, 0.0
MOVR   0.0, 冷却电机速度:VD88
Network 88
LDR>   冷却电机速度:VD88, 30.0
MOVR   25.0, 冷却电机速度:VD88
Network 89
// 初始化下料伺服电机电机速度
LD     恢复出厂设置:V1.7
EU
MOVR   25.0, ROM下料电机速度:VD1740
Network 90
LD     First_Scan_On:SM0.1
MOVR   ROM下料电机速度:VD1740, 下料电机速度:VD128
Network 91
// 将当前值存到ROM区
LD     参数存到ROM:V1605.4
MOVR   下料电机速度:VD128, ROM下料电机速度:VD1740
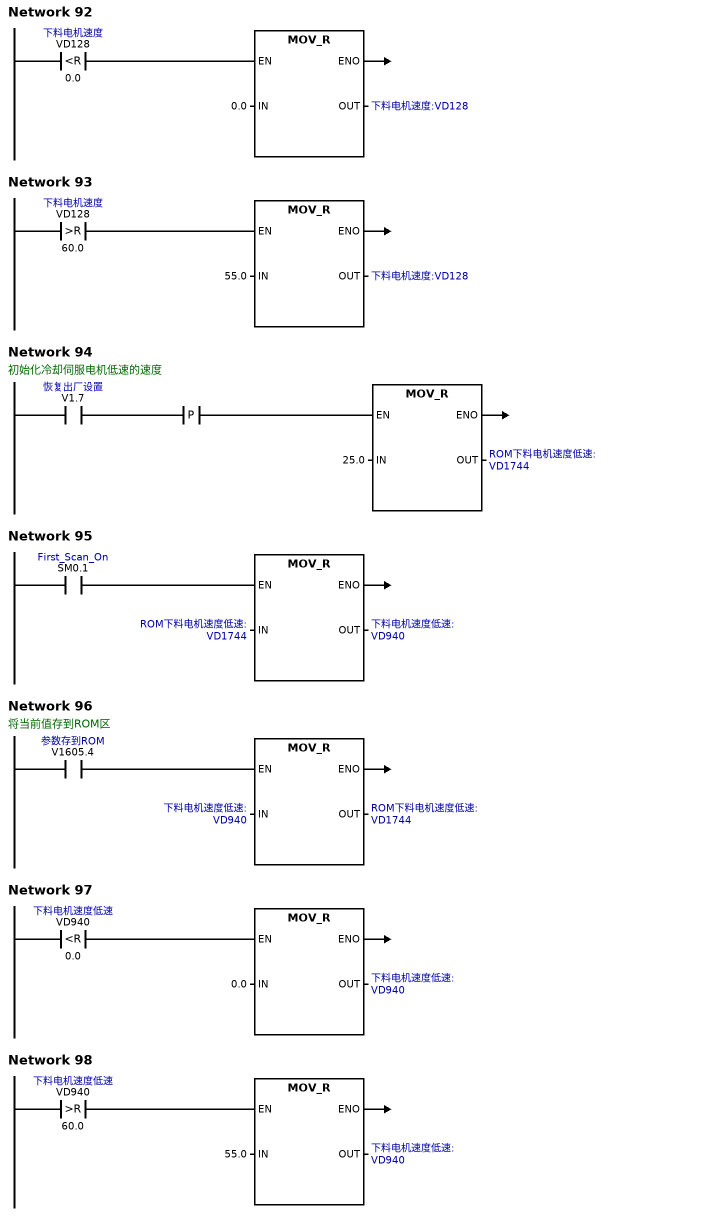
Network 92
LDR<   下料电机速度:VD128, 0.0
MOVR   0.0, 下料电机速度:VD128
Network 93
LDR>   下料电机速度:VD128, 60.0
MOVR   55.0, 下料电机速度:VD128
Network 94
// 初始化冷却伺服电机低速的速度
LD     恢复出厂设置:V1.7
EU
MOVR   25.0, ROM下料电机速度低速:VD1744
Network 95
LD     First_Scan_On:SM0.1
MOVR   ROM下料电机速度低速:VD1744, 下料电机速度低速:VD940
Network 96
// 将当前值存到ROM区
LD     参数存到ROM:V1605.4
MOVR   下料电机速度低速:VD940, ROM下料电机速度低速:VD1744
Network 97
LDR<   下料电机速度低速:VD940, 0.0
MOVR   0.0, 下料电机速度低速:VD940
Network 98
LDR>   下料电机速度低速:VD940, 60.0
MOVR   55.0, 下料电机速度低速:VD940
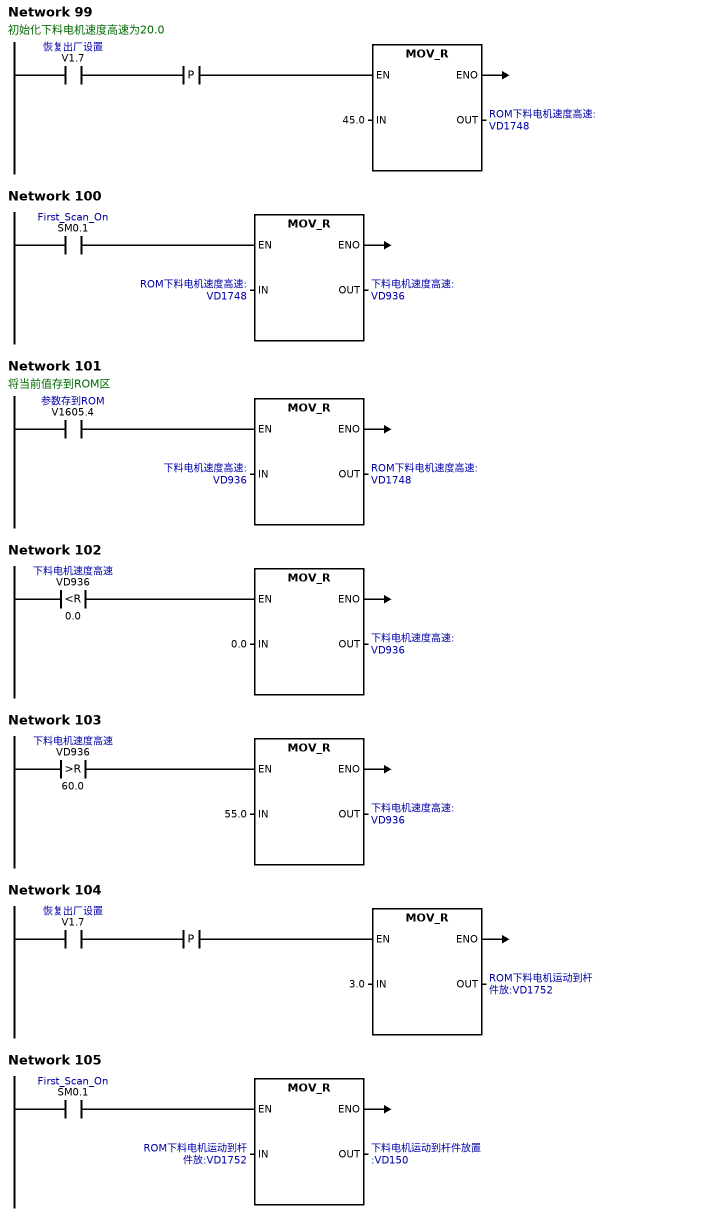
Network 99
// 初始化下料电机速度高速为20.0
LD     恢复出厂设置:V1.7
EU
MOVR   45.0, ROM下料电机速度高速:VD1748
Network 100
LD     First_Scan_On:SM0.1
MOVR   ROM下料电机速度高速:VD1748, 下料电机速度高速:VD936
Network 101
// 将当前值存到ROM区
LD     参数存到ROM:V1605.4
MOVR   下料电机速度高速:VD936, ROM下料电机速度高速:VD1748
Network 102
LDR<   下料电机速度高速:VD936, 0.0
MOVR   0.0, 下料电机速度高速:VD936
Network 103
LDR>   下料电机速度高速:VD936, 60.0
MOVR   55.0, 下料电机速度高速:VD936
Network 104
LD     恢复出厂设置:V1.7
EU
MOVR   3.0, ROM下料电机运动到杆件放:VD1752
Network 105
LD     First_Scan_On:SM0.1
MOVR   ROM下料电机运动到杆件放:VD1752, 下料电机运动到杆件放置:VD150
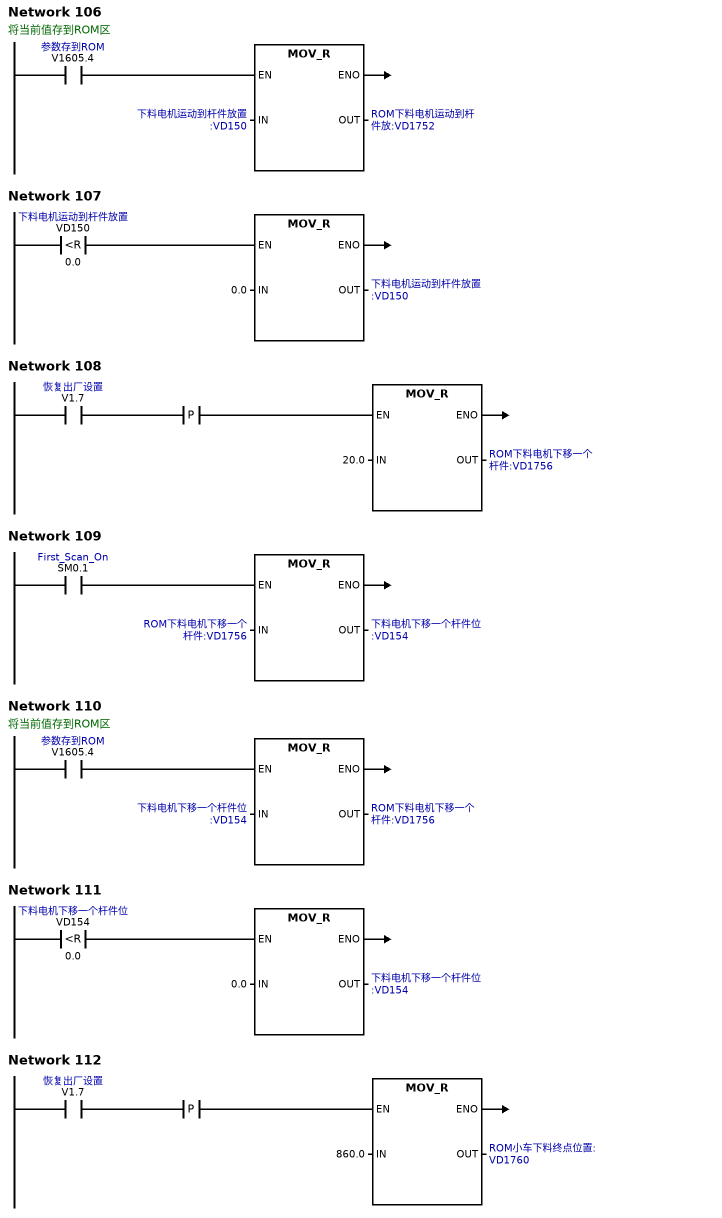
Network 106
// 将当前值存到ROM区
LD     参数存到ROM:V1605.4
MOVR   下料电机运动到杆件放置:VD150, ROM下料电机运动到杆件放:VD1752
Network 107
LDR<   下料电机运动到杆件放置:VD150, 0.0
MOVR   0.0, 下料电机运动到杆件放置:VD150
Network 108
LD     恢复出厂设置:V1.7
EU
MOVR   20.0, ROM下料电机下移一个杆件:VD1756
Network 109
LD     First_Scan_On:SM0.1
MOVR   ROM下料电机下移一个杆件:VD1756, 下料电机下移一个杆件位:VD154
Network 110
// 将当前值存到ROM区
LD     参数存到ROM:V1605.4
MOVR   下料电机下移一个杆件位:VD154, ROM下料电机下移一个杆件:VD1756
Network 111
LDR<   下料电机下移一个杆件位:VD154, 0.0
MOVR   0.0, 下料电机下移一个杆件位:VD154
Network 112
LD     恢复出厂设置:V1.7
EU
MOVR   860.0, ROM小车下料终点位置:VD1760
